// TIA Portal V19 export
TYPE "InfeedAlr"
// stored: Access Published
   STRUCT
      InfeedFault : Bool;   // Fault from infeed telegram
      ComunicationFault : Bool;   // Communication fault from SinaInfeed
      TimeoutActivation : Bool;   // Timeout infeed running
      GeneralError : Bool;   // General error from SinaInfeed
   END_STRUCT;
END_TYPE
